Staubli VAL3: CREATDIR.pgx

public program CreatDir(string x_sDirName (dimensions=1), bool& x_bRes (dimensions=1))
  local num l_nFileID
begin
  //说明：x_sDirName一般为 /usr/usrapp
  //
  //



  x_bRes=false
  //目录名为空则返回
  if x_sDirName==""
    return
  endIf

  //打开文件，如果文件不存在则新建文件
  l_nFileID=$fileOpen(x_sDirName+"\text","w")
  if l_nFileID<0 or l_nFileID>9
    return
  endIf
  //关闭文件
  call CloseFile(l_nFileID)
  //删除文件  保留目录
  $delete(x_sDirName+"\text")
  x_bRes=true


end
